FUNCTION_BLOCK CM_TubeLedRgb IMPLEMENTS I_LedRgb

VAR_INPUT
	i_ref_eCtrlMode : REFERENCE TO E_CtrlMode;
	i_ref_eCtrlState : REFERENCE TO E_CtrlState;
END_VAR

VAR
	//Outputs
	Q_bColorRed AT %Q* : BOOL;
	Q_bColorGreen AT %Q* : BOOL;
	Q_bColorBlue AT %Q* : BOOL;
	Q_bColorWhite AT %Q* : BOOL;
	
	// Force outputs (IO-test functions)
	s_fbForceLedTubeRed : FB_ForceOutput;
	s_fbForceLedTubeGreen : FB_ForceOutput;
	s_fbForceLedTubeBlue : FB_ForceOutput;
	s_fbForceLedTubeWhite : FB_ForceOutput;
	
	//Variables
	s_bColorRed : BOOL;
	s_bColorGreen : BOOL;
	s_bColorBlue : BOOL;
	s_bColorWhite : BOOL;
	s_nStaColor : BYTE; //Binairy code RGBW
	
	//Commands
	s_bCmdColorRed : BOOL;
	s_bCmdColorGreen : BOOL;
	s_bCmdColorBlue : BOOL;
	s_bCmdColorWhite : BOOL;
	
	s_bFlash : BOOL;
	s_fbFlash : FB_Flash;
END_VAR


s_fbFlash(
	i_bExcecute := TRUE,
	t_tOnTime := T#750MS,
	t_tOffTime := T#750MS);
	
IF s_bFlash THEN
	s_bCmdColorRed := s_bColorRed AND s_fbFlash.o_bQ;
	s_bCmdColorGreen := s_bColorGreen AND s_fbFlash.o_bQ;
	s_bCmdColorBlue := s_bColorBlue AND s_fbFlash.o_bQ;
	s_bCmdColorWhite := s_bColorWhite AND s_fbFlash.o_bQ;
ELSE
	s_bCmdColorRed := s_bColorRed;
	s_bCmdColorGreen := s_bColorGreen;
	s_bCmdColorBlue := s_bColorBlue;
	s_bCmdColorWhite := s_bColorWhite;
END_IF

{warning #TODO: Nog bepalen OF het beter is om onderstaande code te verwerken in FB_Force output}
IF __ISVALIDREF(i_ref_eCtrlMode) AND __ISVALIDREF(i_ref_eCtrlState) THEN
	IF (i_ref_eCtrlMode <> E_CtrlMode.IO) OR (i_ref_eCtrlState <> E_CtrlState.RUNNING) THEN
		s_fbForceLedTubeRed.i_eForceValue := E_ForceValue.RELEASED;
		s_fbForceLedTubeGreen.i_eForceValue := E_ForceValue.RELEASED;
		s_fbForceLedTubeBlue.i_eForceValue := E_ForceValue.RELEASED;
		s_fbForceLedTubeWhite.i_eForceValue := E_ForceValue.RELEASED;
	END_IF
END_IF 

//Force RGB-outputs FALSE if W-output is TRUE
IF Q_bColorWhite THEN
	s_fbForceLedTubeRed.i_eForceValue := E_ForceValue.FORCE_OFF;
	s_fbForceLedTubeGreen.i_eForceValue := E_ForceValue.FORCE_OFF;
	s_fbForceLedTubeBlue.i_eForceValue := E_ForceValue.FORCE_OFF;
END_IF

//Force W-output FALSE if any RGB-output is TRUE
IF Q_bColorRed OR Q_bColorGreen OR Q_bColorBlue THEN
	s_fbForceLedTubeWhite.i_eForceValue := E_ForceValue.FORCE_OFF;
END_IF

s_fbForceLedTubeRed(
	i_ref_bCmdInput := s_bCmdColorRed,
	i_ref_bCmdOutput := Q_bColorRed);
	
s_fbForceLedTubeGreen(
	i_ref_bCmdInput := s_bCmdColorGreen,
	i_ref_bCmdOutput := Q_bColorGreen);
	
s_fbForceLedTubeBlue(
	i_ref_bCmdInput := s_bCmdColorBlue,
	i_ref_bCmdOutput := Q_bColorBlue);
	
s_fbForceLedTubeWhite(
	i_ref_bCmdInput := s_bCmdColorWhite,
	i_ref_bCmdOutput := Q_bColorWhite);

METHOD PUBLIC m_Blue : BOOL
VAR_INPUT
	i_bFlash : BOOL;
END_VAR

s_bColorRed := FALSE;
s_bColorGreen := FALSE;
s_bColorBlue := TRUE;
s_bColorWhite := FALSE;
s_nStaColor := 4;

s_bFlash := i_bFlash;
END_METHOD

METHOD PUBLIC m_Cyan : BOOL
VAR_INPUT
	i_bFlash : BOOL;
END_VAR

s_bColorRed := FALSE;
s_bColorGreen := TRUE;
s_bColorBlue := TRUE;
s_bColorWhite := FALSE;
s_nStaColor := 6;

s_bFlash := i_bFlash;
END_METHOD

METHOD PUBLIC m_Green : BOOL
VAR_INPUT
	i_bFlash : BOOL;
END_VAR

s_bColorRed := FALSE;
s_bColorGreen := TRUE;
s_bColorBlue := FALSE;
s_bColorWhite := FALSE;
s_nStaColor := 2;

s_bFlash := i_bFlash;
END_METHOD

METHOD PUBLIC m_Magenta : BOOL
VAR_INPUT
	i_bFlash : BOOL;
END_VAR

s_bColorRed := TRUE;
s_bColorGreen := FALSE;
s_bColorBlue := TRUE;
s_bColorWhite := FALSE;
s_nStaColor := 5;

s_bFlash := i_bFlash;
END_METHOD

METHOD PUBLIC m_Off : BOOL
VAR_INPUT
	i_bFlash : BOOL;
END_VAR

s_bColorRed := FALSE;
s_bColorGreen := FALSE;
s_bColorBlue := FALSE;
s_bColorWhite := FALSE;
s_nStaColor := 0;

s_bFlash := i_bFlash;
END_METHOD

METHOD PUBLIC m_Red : BOOL
VAR_INPUT
	i_bFlash : BOOL;
END_VAR

s_bColorRed := TRUE;
s_bColorGreen := FALSE;
s_bColorBlue := FALSE;
s_bColorWhite := FALSE;
s_nStaColor := 1;

s_bFlash := i_bFlash;
END_METHOD

METHOD PUBLIC m_White : BOOL
VAR_INPUT
	i_bFlash : BOOL;
END_VAR

s_bColorRed := FALSE;
s_bColorGreen := FALSE;
s_bColorBlue := FALSE;
s_bColorWhite := TRUE;
s_nStaColor := 8;

s_bFlash := i_bFlash;
END_METHOD

METHOD PUBLIC m_Yellow : BOOL
VAR_INPUT
	i_bFlash : BOOL;
END_VAR

s_bColorRed := TRUE;
s_bColorGreen := TRUE;
s_bColorBlue := FALSE;
s_bColorWhite := FALSE;
s_nStaColor := 3;

s_bFlash := i_bFlash;
END_METHOD

{attribute 'monitoring':='call'}
PROPERTY PUBLIC p_bStaColorBlue : BOOL
GET

p_bStaColorBlue := Q_bColorBlue;
END_GET
END_PROPERTY

{attribute 'monitoring':='call'}
PROPERTY PUBLIC p_bStaColorGreen : BOOL
GET

p_bStaColorGreen := Q_bColorGreen;
END_GET
END_PROPERTY

{attribute 'monitoring':='call'}
PROPERTY PUBLIC p_bStaColorRed : BOOL
GET

p_bStaColorRed := Q_bColorRed;
END_GET
END_PROPERTY

{attribute 'monitoring':='call'}
PROPERTY PUBLIC p_bStaColorWhite : BOOL
GET

p_bStaColorWhite := Q_bColorWhite;
END_GET
END_PROPERTY

{attribute 'monitoring':='call'}
PROPERTY PUBLIC p_nStaColor : BYTE //Binairy code RGBW
GET

p_nStaColor := s_nStaColor;
END_GET
END_PROPERTY

END_FUNCTION_BLOCK

(* stored: Version 1.1.0.1, ProductVersion 3.1.4024.12
   POU CM_TubeLedRgb: Id {595df5ed-8c43-4c64-84d2-9ba9d4b953e6}, SpecialFunc None
   Method m_Blue: Id {d57b0497-a91a-4eae-8ab3-33ff974915fa}
   Method m_Cyan: Id {fe6a9e1a-de65-436f-b497-7fc6b195b9fe}
   Method m_Green: Id {5b8239f4-a47d-49ab-b71e-dde0e6e7a3a2}
   Method m_Magenta: Id {6a1891b6-ba70-4e68-82c9-b34683cfce47}
   Method m_Off: Id {ecf7c0ec-aeb1-4f25-9b33-59f6fa463870}
   Method m_Red: Id {97ed4e1e-4f76-4552-9da8-d9193d17516b}
   Method m_White: Id {290105c0-46ae-4f2f-9dea-cc91419b9a9c}
   Method m_Yellow: Id {b5d6329c-fb65-418c-8370-735d2a6d1618}
   Property p_bStaColorBlue: Id {088d2652-fedb-418c-9294-37610dda26a0}
   Get Get: Id {7bd8b468-a96f-43cf-a618-1b1ada3749d7}
   Property p_bStaColorGreen: Id {5eec6bb9-a994-4c2c-9e57-0a28e72f2f1f}
   Get Get: Id {84208be1-5d3e-4a65-b236-f8c77fde461a}
   Property p_bStaColorRed: Id {2ff5d3e0-4676-4b93-890d-eb205211f9cc}
   Get Get: Id {87fafabc-0fa0-4802-be84-5a31e59deb5a}
   Property p_bStaColorWhite: Id {1c67a4bc-70c9-4b89-a889-b5e68a56771a}
   Get Get: Id {ba22e263-dca3-4b7a-990e-31799bde4927}
   Property p_nStaColor: Id {16cca93e-023e-4a33-82d3-73facd1cf405}
   Get Get: Id {374cfdc8-85e5-4ebd-a15d-cbe78fc6fbaf} *)
